FUNCTION FUN_AX5000_GetMainVoltageUINT : UINT
VAR_INPUT
		Axis									:	Tc2_Mc2.AXIS_REF;
END_VAR
VAR
		SoERead 								:	Tc2_Mc2_Drive.FB_SoERead;
		SoEReadValue 							:	UINT;
		Busy									:	BOOL;
END_VAR

// AX5000 Get Mains Voltage
// This block is made for inspirational purposes.
// Please make your own version that complies with your / your company´s programming vision
// Version 1.0 - Initial Version
//-----------------------------------------------------------------------------------------

IF NOT SoERead.Busy AND busy THEN
	IF NOT SoERead.error THEN
		FUN_AX5000_GetMainVoltageUINT := SoEReadValue;
	END_IF
END_IF
SoERead(Axis:=Axis,Element:=16#40,pDstBuf:=ADR(SoEReadValue),BufLen:=SIZEOF(SoEReadValue));
SoERead.Idn := P_0_IDNs + 217; 
SoERead.Execute := TRUE;
IF SoERead.Busy THEN
	Busy :=1;
END_IF

END_FUNCTION

(* stored: Version 1.1.0.1, ProductVersion 3.1.4024.14
   POU FUN_AX5000_GetMainVoltageUINT: Id {67adc20e-4ce4-4904-91c0-489276e25e98}, SpecialFunc None *)
